(* CODESYS project Esteira Contadora de Caixas.project

Project tree, tasks and I/O mapping:
  Device : CODESYS Control Win V3, 3S - Smart Software Solutions GmbH, order no. 305021, version 3.5.11.30
    application Application
      libraries: Standard, * (System)
      task MainTask (cyclic, interval t#20ms, priority 1) calls PLC_PRG
      program PLC_PRG [LD]
      Symbols
*)

// Device/Application/PLC_PRG
PROGRAM PLC_PRG
VAR
	Sirene:BOOL;
	LED_Alerta:BOOL;
	LED_Ligado:BOOL;
	LED_Desligado:BOOL;
	Reset:BOOL;
	Start:BOOL;
	Stop:BOOL;
	Contagem:INT;
	Emergencia:BOOL; 
	Sensor_S1:BOOL;
	Sensor_S2:BOOL;
	Sensor_S3:BOOL;
	Esteira1:BOOL;
	Esteira2:BOOL;
	M1:BOOL;
	
	CTU_0: CTU;
	TON_0: TON;
END_VAR
VAR // added by the converter: edge detectors and wires of the graphical bodies
    _w1 : BOOL;
    _rt1 : R_TRIG;
END_VAR

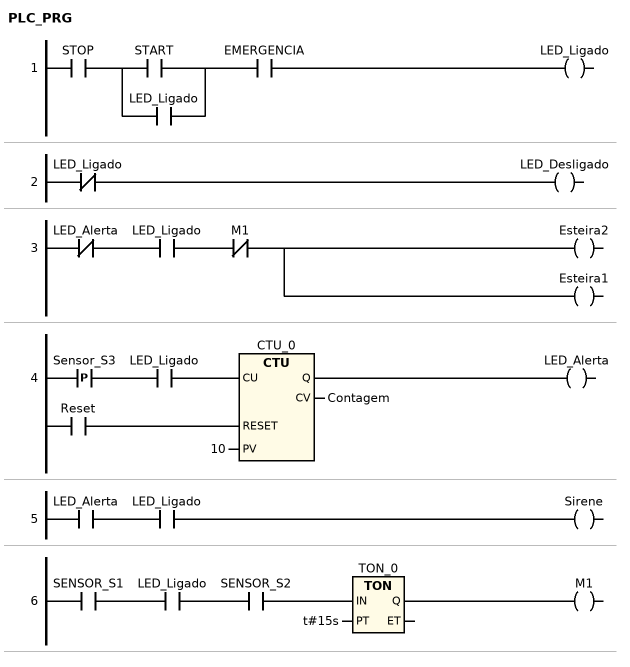
// NETWORK 1
LED_Ligado := STOP AND (START OR LED_Ligado) AND EMERGENCIA;

// NETWORK 2
LED_Desligado := NOT LED_Ligado;

// NETWORK 3
_w1 := NOT LED_Alerta AND LED_Ligado AND NOT M1;
Esteira2 := _w1;
Esteira1 := _w1;

// NETWORK 4
_rt1(CLK := Sensor_S3);
CTU_0(CU := _rt1.Q AND LED_Ligado, RESET := Reset, PV := 10, CV => Contagem); // CTU
LED_Alerta := CTU_0.Q;

// NETWORK 5
Sirene := LED_Alerta AND LED_Ligado;

// NETWORK 6
TON_0(IN := SENSOR_S1 AND LED_Ligado AND SENSOR_S2, PT := t#15s); // TON
M1 := TON_0.Q;

END_PROGRAM
